FUNCTION_BLOCK FB_DataHistory_Real
VAR_INPUT
	_val : REAL;
	_save : BOOL;
END_VAR
VAR_OUTPUT
	_array : ARRAY [0.._history] OF REAL;
END_VAR
VAR
	_i : INT;
END_VAR

IF _save THEN
	FOR _i := 0 TO _history - 1 DO
		_array[_i] := _array[_i + 1];
	END_FOR
	_array[_history] := _val;
END_IF

END_FUNCTION_BLOCK

(* stored: Version 1.1.0.1, ProductVersion 3.1.4018.5
   POU FB_DataHistory_Real: Id {a54ca4a3-be42-49d7-af9f-454ee6d36173}, SpecialFunc None *)
